TYPE FRACTION :
STRUCT
	NUMERATOR : INT;
	DENOMINATOR : INT;
END_STRUCT
END_TYPE

(* stored: Version 1.1.0.1, ProductVersion 3.1.4022.7
   DUT FRACTION: Id {f2e0f826-af7c-4d6b-b45f-c853f0dd1efc} *)
